// TIA Portal V16 export
// export: Created 2023-06-21T17:06:27.8351272Z, ExportSetting WithDefaults, DisplayName Totally Integrated Automation Portal, DisplayVersion V16 Update 4, DisplayName TIA Portal Version Control Interface, DisplayVersion V16 Update 2, DisplayName TIA Portal Openness, DisplayVersion V16 Update 4, DisplayName SINAMICS Startdrive Advanced, DisplayVersion V16, DisplayName SINAMICS Startdrive G130, G150, S120, S150, SINAMICS MV, S210, DisplayVersion V16, DisplayName SINAMICS Startdrive G110M, G120, G120C, G120D, G120P, DisplayVersion V16, DisplayName STEP 7 Professional, DisplayVersion V16 Update 4, DisplayName STEP 7 Safety, DisplayVersion V16, DisplayName Soft Starter ES, DisplayVersion V16, DisplayName WinCC Advanced, DisplayVersion V16 Update 4
DATA_BLOCK "Modbus_Master_DB"   // DB3
// stored: AutoNumber true, DBAccessibleFromOPCUA true, InstanceOfName Modbus_Master, OfSystemLibElement Modbus_Master, OfSystemLibVersion 3.3
"Modbus_Master"
   // VAR_INPUT
   //    REQ : Bool;
   //    MB_ADDR : UInt;
   //    MODE : USInt;
   //    DATA_ADDR : UDInt;
   //    DATA_LEN : UInt;
   // END_VAR
   // VAR_OUTPUT
   //    DONE : Bool;
   //    BUSY : Bool;
   //    ERROR : Bool;
   //    STATUS : Word;
   // END_VAR
   // VAR_IN_OUT
   //    DATA_PTR : Variant;
   // END_VAR
   // VAR
   //    MB_State : SInt;
   //    Blocked_Proc_Timeout : Real;
   //    Extended_Addressing : Bool;
   //    Compatibility_Mode : Bool;
   //    MB_DB { S7_SetPoint := 'True'} : P2P_MB_BASE;
   //    Send_P2P { S7_SetPoint := 'True'} : Send_P2P;
   //    Receive_P2P { S7_SetPoint := 'True'} : Receive_P2P;
   //    Receive_Reset { S7_SetPoint := 'True'} : Receive_Reset;
   //    S_PORT : Word;
   //    S_RESP_TO : Word;
   //    S_ICHAR_GAP : Word;
   //    S_RETRIES : Word;
   //    S_MB_ADDR : UInt;
   //    S_MODE : USInt;
   //    S_DATA_ADDR : UDInt;
   //    S_DATA_LEN : UInt;
   //    w_retries : Word;
   //    y_SlaveAddrHi : Byte;
   //    y_SlaveAddrLo : Byte;
   //    StartAddress : Word;
   //    Value : Word;
   //    y_FCode : Byte;
   //    INTERNAL_CDATA : Array[1..257] of Byte;
   //    mb_timer { S7_SetPoint := 'True'} : TON_TIME;
   //    TimeElapsed : Bool;
   // END_VAR
BEGIN
END_DATA_BLOCK
